// TIA Portal V17 export
// export: Created 2025-03-07T09:18:28.8674734Z, ExportSetting WithDefaults, DisplayName Totally Integrated Automation Portal, DisplayVersion V17 Update 8, DisplayName TIA Portal Openness, DisplayVersion V17 Update 8, DisplayName TIA Portal Version Control Interface, DisplayVersion V17, DisplayName SINAMICS Startdrive Advanced, DisplayVersion V17 SP2, DisplayName SINAMICS Startdrive G110M, G120, G120C, G120D, G120P, G115D, DisplayVersion V17 SP2, DisplayName SINAMICS Startdrive G130, G150, S120, S150, SINAMICS MV, S210, DisplayVersion V17 SP2, DisplayName STEP 7 Professional, DisplayVersion V17 Update 8, DisplayName SINUMERIK ONE STEP 7 Toolbox, DisplayVersion V17 Update 12, DisplayName SINUMERIK 840D sl STEP 7 Toolbox, DisplayVersion V17 Update 12, DisplayName STEP 7 Safety, DisplayVersion V17 Update 6, DisplayName WinCC Advanced, DisplayVersion V17 Update 8
FUNCTION "UPTL_InitialiseConfigData" : Void   // FC1050, LAD
{ S7_Optimized_Access := 'FALSE' }
AUTHOR : Transline
FAMILY : UPTL_Transline
VERSION : 4.0
// stored: AutoNumber true, IsIECCheckEnabled false, SetENOAutomatically false, UDAEnableTagReadback false
   VAR CONSTANT
      "CONST_Local~Interface" : HW_INTERFACE := 266;
   END_VAR
BEGIN

REGION Network 1
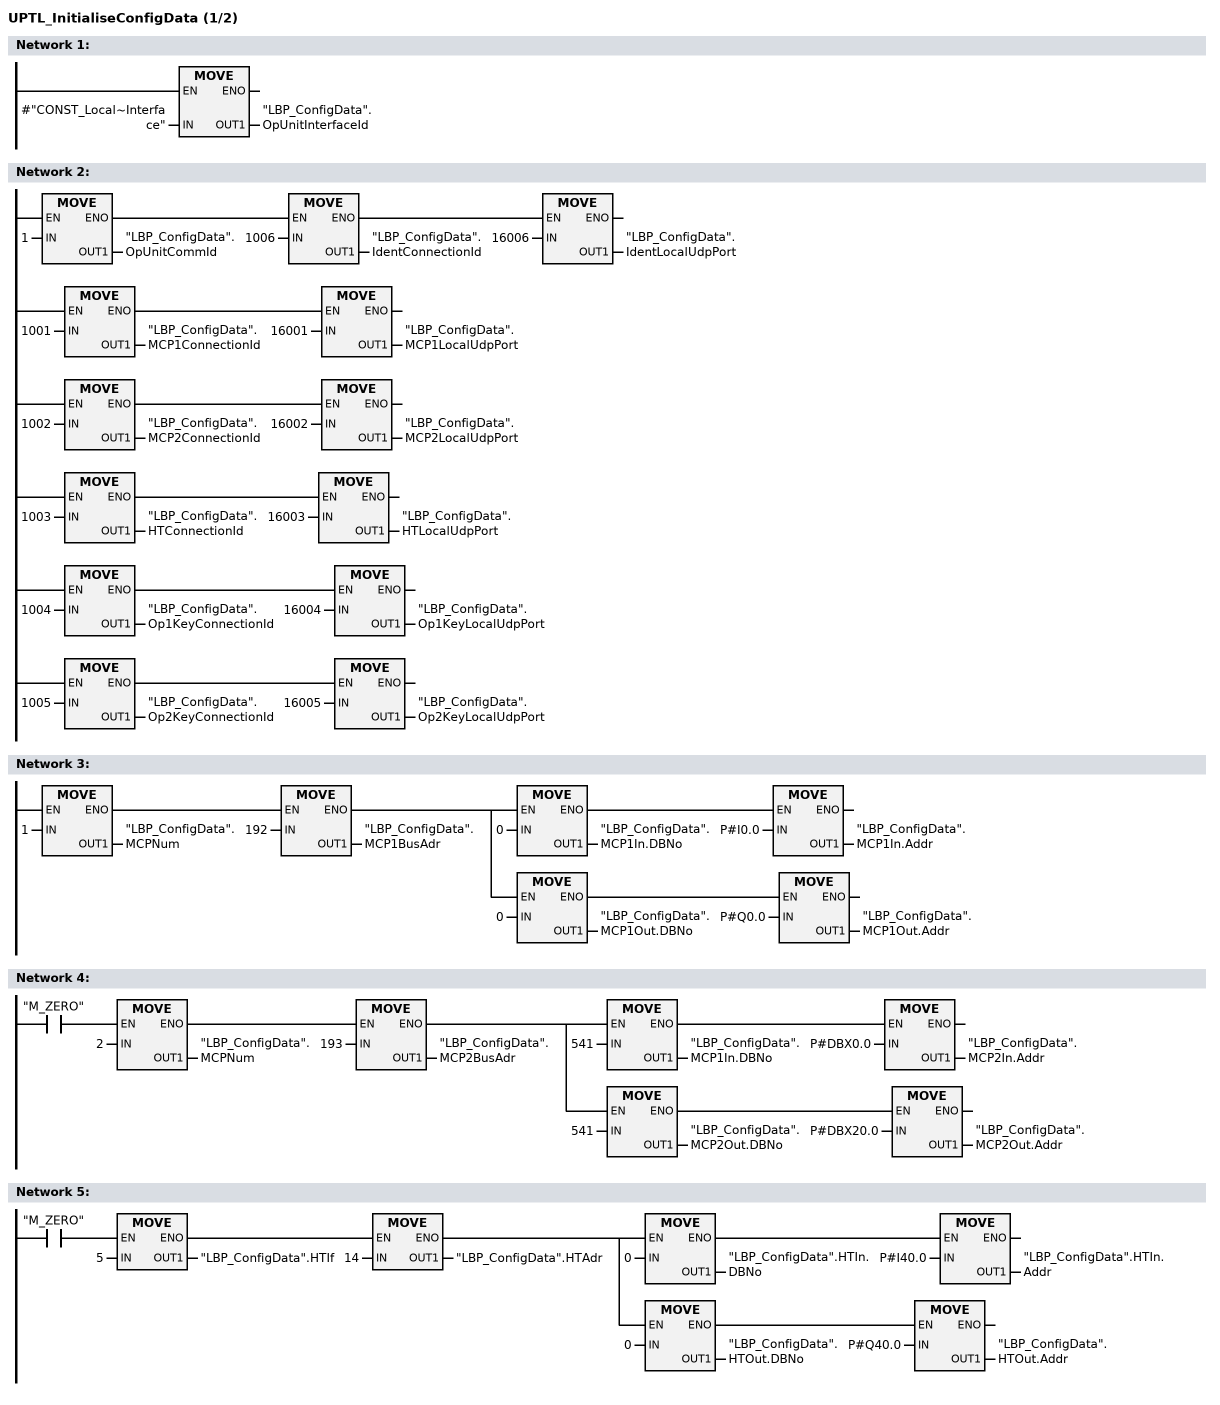
   RUNG wire#powerrail
      Move(in := #"CONST_Local~Interface", out1 => "LBP_ConfigData".OpUnitInterfaceId)
   END_RUNG
   // the same network as SCL:
   "LBP_ConfigData".OpUnitInterfaceId := #"CONST_Local~Interface";
END_REGION

REGION Network 2
   RUNG wire#powerrail
      Move(in := 1, out1 => "LBP_ConfigData".OpUnitCommId)
      Move(in := 1006, out1 => "LBP_ConfigData".IdentConnectionId)
      Move(in := 16006, out1 => "LBP_ConfigData".IdentLocalUdpPort)
   END_RUNG
   RUNG wire#powerrail
      Move(in := 1001, out1 => "LBP_ConfigData".MCP1ConnectionId)
      Move(in := 16001, out1 => "LBP_ConfigData".MCP1LocalUdpPort)
   END_RUNG
   RUNG wire#powerrail
      Move(in := 1002, out1 => "LBP_ConfigData".MCP2ConnectionId)
      Move(in := 16002, out1 => "LBP_ConfigData".MCP2LocalUdpPort)
   END_RUNG
   RUNG wire#powerrail
      Move(in := 1003, out1 => "LBP_ConfigData".HTConnectionId)
      Move(in := 16003, out1 => "LBP_ConfigData".HTLocalUdpPort)
   END_RUNG
   RUNG wire#powerrail
      Move(in := 1004, out1 => "LBP_ConfigData".Op1KeyConnectionId)
      Move(in := 16004, out1 => "LBP_ConfigData".Op1KeyLocalUdpPort)
   END_RUNG
   RUNG wire#powerrail
      Move(in := 1005, out1 => "LBP_ConfigData".Op2KeyConnectionId)
      Move(in := 16005, out1 => "LBP_ConfigData".Op2KeyLocalUdpPort)
   END_RUNG
   // the same network as SCL:
   "LBP_ConfigData".OpUnitCommId := 1;
   "LBP_ConfigData".IdentConnectionId := 1006;
   "LBP_ConfigData".IdentLocalUdpPort := 16006;
   "LBP_ConfigData".MCP1ConnectionId := 1001;
   "LBP_ConfigData".MCP1LocalUdpPort := 16001;
   "LBP_ConfigData".MCP2ConnectionId := 1002;
   "LBP_ConfigData".MCP2LocalUdpPort := 16002;
   "LBP_ConfigData".HTConnectionId := 1003;
   "LBP_ConfigData".HTLocalUdpPort := 16003;
   "LBP_ConfigData".Op1KeyConnectionId := 1004;
   "LBP_ConfigData".Op1KeyLocalUdpPort := 16004;
   "LBP_ConfigData".Op2KeyConnectionId := 1005;
   "LBP_ConfigData".Op2KeyLocalUdpPort := 16005;
END_REGION

REGION Network 3
   RUNG wire#powerrail
      Move(in := 1, out1 => "LBP_ConfigData".MCPNum)
      Move(in := 192, out1 => "LBP_ConfigData".MCP1BusAdr)
      wire#w1
      Move(in := 0, out1 => "LBP_ConfigData".MCP1In.DBNo)
      Move(in := P#I0.0, out1 => "LBP_ConfigData".MCP1In.Addr)
   END_RUNG
   RUNG wire#w1
      Move(in := 0, out1 => "LBP_ConfigData".MCP1Out.DBNo)
      Move(in := P#Q0.0, out1 => "LBP_ConfigData".MCP1Out.Addr)
   END_RUNG
   // the same network as SCL:
   "LBP_ConfigData".MCPNum := 1;
   "LBP_ConfigData".MCP1BusAdr := 192;
   "LBP_ConfigData".MCP1In.DBNo := 0;
   "LBP_ConfigData".MCP1In.Addr := P#I0.0;
   "LBP_ConfigData".MCP1Out.DBNo := 0;
   "LBP_ConfigData".MCP1Out.Addr := P#Q0.0;
END_REGION

REGION Network 4
   RUNG wire#powerrail
      Contact( "M_ZERO" )
      Move(in := 2, out1 => "LBP_ConfigData".MCPNum)
      Move(in := 193, out1 => "LBP_ConfigData".MCP2BusAdr)
      wire#w1
      Move(in := 541, out1 => "LBP_ConfigData".MCP1In.DBNo)
      Move(in := P#DBX0.0, out1 => "LBP_ConfigData".MCP2In.Addr)
   END_RUNG
   RUNG wire#w1
      Move(in := 541, out1 => "LBP_ConfigData".MCP2Out.DBNo)
      Move(in := P#DBX20.0, out1 => "LBP_ConfigData".MCP2Out.Addr)
   END_RUNG
   // the same network as SCL:
   IF "M_ZERO" THEN
       "LBP_ConfigData".MCPNum := 2;
       "LBP_ConfigData".MCP2BusAdr := 193;
       "LBP_ConfigData".MCP1In.DBNo := 541;
       "LBP_ConfigData".MCP2In.Addr := P#DBX0.0;
       "LBP_ConfigData".MCP2Out.DBNo := 541;
       "LBP_ConfigData".MCP2Out.Addr := P#DBX20.0;
   END_IF;
END_REGION

REGION Network 5
   RUNG wire#powerrail
      Contact( "M_ZERO" )
      Move(in := 5, out1 => "LBP_ConfigData".HTIf)
      Move(in := 14, out1 => "LBP_ConfigData".HTAdr)
      wire#w1
      Move(in := 0, out1 => "LBP_ConfigData".HTIn.DBNo)
      Move(in := P#I40.0, out1 => "LBP_ConfigData".HTIn.Addr)
   END_RUNG
   RUNG wire#w1
      Move(in := 0, out1 => "LBP_ConfigData".HTOut.DBNo)
      Move(in := P#Q40.0, out1 => "LBP_ConfigData".HTOut.Addr)
   END_RUNG
   // the same network as SCL:
   IF "M_ZERO" THEN
       "LBP_ConfigData".HTIf := 5;
       "LBP_ConfigData".HTAdr := 14;
       "LBP_ConfigData".HTIn.DBNo := 0;
       "LBP_ConfigData".HTIn.Addr := P#I40.0;
       "LBP_ConfigData".HTOut.DBNo := 0;
       "LBP_ConfigData".HTOut.Addr := P#Q40.0;
   END_IF;
END_REGION

REGION Network 6
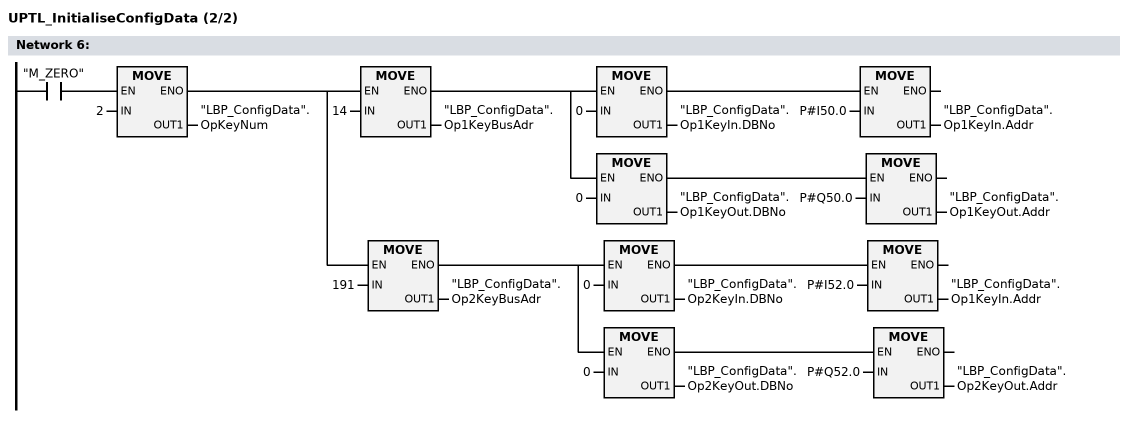
   RUNG wire#powerrail
      Contact( "M_ZERO" )
      Move(in := 2, out1 => "LBP_ConfigData".OpKeyNum)
      wire#w1
      Move(in := 14, out1 => "LBP_ConfigData".Op1KeyBusAdr)
      wire#w2
      Move(in := 0, out1 => "LBP_ConfigData".Op1KeyIn.DBNo)
      Move(in := P#I50.0, out1 => "LBP_ConfigData".Op1KeyIn.Addr)
   END_RUNG
   RUNG wire#w2
      Move(in := 0, out1 => "LBP_ConfigData".Op1KeyOut.DBNo)
      Move(in := P#Q50.0, out1 => "LBP_ConfigData".Op1KeyOut.Addr)
   END_RUNG
   RUNG wire#w1
      Move(in := 191, out1 => "LBP_ConfigData".Op2KeyBusAdr)
      wire#w3
      Move(in := 0, out1 => "LBP_ConfigData".Op2KeyIn.DBNo)
      Move(in := P#I52.0, out1 => "LBP_ConfigData".Op1KeyIn.Addr)
   END_RUNG
   RUNG wire#w3
      Move(in := 0, out1 => "LBP_ConfigData".Op2KeyOut.DBNo)
      Move(in := P#Q52.0, out1 => "LBP_ConfigData".Op2KeyOut.Addr)
   END_RUNG
   // the same network as SCL:
   IF "M_ZERO" THEN
       "LBP_ConfigData".OpKeyNum := 2;
       "LBP_ConfigData".Op1KeyBusAdr := 14;
       "LBP_ConfigData".Op1KeyIn.DBNo := 0;
       "LBP_ConfigData".Op1KeyIn.Addr := P#I50.0;
       "LBP_ConfigData".Op1KeyOut.DBNo := 0;
       "LBP_ConfigData".Op1KeyOut.Addr := P#Q50.0;
       "LBP_ConfigData".Op2KeyBusAdr := 191;
       "LBP_ConfigData".Op2KeyIn.DBNo := 0;
       "LBP_ConfigData".Op1KeyIn.Addr := P#I52.0;
       "LBP_ConfigData".Op2KeyOut.DBNo := 0;
       "LBP_ConfigData".Op2KeyOut.Addr := P#Q52.0;
   END_IF;
END_REGION
END_FUNCTION
